// TIA Portal V21 export
FUNCTION_BLOCK "SwitchgearSim"   // FB6, FBD
{ S7_Optimized_Access := 'TRUE' }
// stored: MemoryReserve 100, SetENOAutomatically false
   VAR_INPUT
      start : Bool;
      stop : Bool;
      opCurrent : LReal;
      "dt" : Time;
      notReadyFlt : Bool;
      resetBlock : Bool;
   END_VAR
   VAR_OUTPUT
      readySg : Bool;
      fbOn : Bool;
      fbOff : Bool;
      current : Real;
   END_VAR
   VAR
      onTimer : TON_TIME;
      offTimer : TON_TIME;
      currentFOTD { S7_SetPoint := 'True'} : "Fotd";
   END_VAR
   VAR_TEMP   // added for the SCL form of the ladder/FBD networks
      _w1 : Bool;
   END_VAR
BEGIN

REGION Network 1
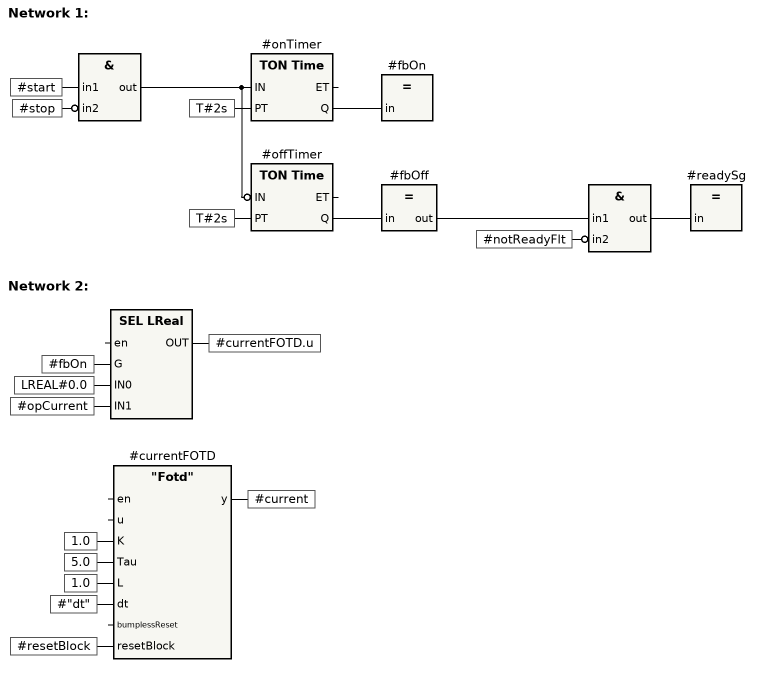
   #_w1 := #start AND NOT #stop;
   #onTimer(IN := #_w1, PT := T#2s);   // TON
   #fbOn := #onTimer.Q;
   #offTimer(IN := NOT #_w1, PT := T#2s);   // TON
   #fbOff := #offTimer.Q;
   #readySg := #offTimer.Q AND NOT #notReadyFlt;
END_REGION

REGION Network 2
   #currentFOTD.u := SEL(G := #fbOn, IN0 := LREAL#0.0, IN1 := #opCurrent);
   #currentFOTD(K := 1.0, Tau := 5.0, L := 1.0, "dt" := #"dt", resetBlock := #resetBlock, y => #current);   // "Fotd"
END_REGION
END_FUNCTION_BLOCK
